FUNCTION_BLOCK PUBLIC EcMasterDeviceCount IMPLEMENTS IEcTask
VAR_INPUT
END_VAR
VAR_OUTPUT
END_VAR
VAR
	iState : INT;
	masterDeviceCount : Tc2_EtherCAT.FB_EcGetSlaveCount;
	_execute: BOOL;
	_done: BOOL;
	_busy: BOOL;
	_error: BOOL;
	_netId: AMSNETID;
END_VAR

CASE iState OF
	0:
		IF _execute THEN
			_done := FALSE;
			_busy := TRUE;
			_error := FALSE;
			masterDeviceCount.bExecute := TRUE;
			IF masterDeviceCount.bBusy THEN
				iState := 10;
				_execute := false;
			END_IF
		END_IF
	10:
		IF NOT masterDeviceCount.bBusy THEN
			IF NOT masterDeviceCount.bError THEN
				_done := TRUE;
			ELSE
				_error := TRUE;
			END_IF
			_busy := FALSE;
			masterDeviceCount.bExecute := FALSE;
			iState := 0;
		END_IF
END_CASE

masterDeviceCount(sNetId := Tc2_System.F_CreateAmsNetId(nIds := NetId));

{warning 'add method implementation '}
METHOD Abort : BOOL
masterDeviceCount.bExecute := FALSE;
_busy := FALSE;
_execute := FALSE;
Abort := TRUE;
iState := 0;
END_METHOD

{warning 'add property implementation'}
PROPERTY Busy : BOOL
GET
Busy := _busy;
END_GET
END_PROPERTY

{warning 'add property implementation'}
PROPERTY Done : BOOL
GET
Done := _done;
END_GET
END_PROPERTY

{warning 'add property implementation'}
PROPERTY Error : BOOL
GET
Error := _error;
END_GET
END_PROPERTY

METHOD Execute : BOOL
VAR_INPUT
END_VAR
IF NOT Busy THEN
	Execute := _execute := TRUE;
END_IF
END_METHOD

{warning 'add property implementation'}
PROPERTY NetID : amsnetid
GET
NetID := _netId;
END_GET
SET
_netId := NetID;
END_SET
END_PROPERTY

PROPERTY NumberDevices : uint
GET
NumberDevices := masterDeviceCount.nSlaves;
END_GET
END_PROPERTY

END_FUNCTION_BLOCK

(* stored: Version 1.1.0.1, ProductVersion 3.1.4024.11
   POU EcMasterDeviceCount: Id {fc00524b-5402-4693-86e9-fa947a8c9c97}, SpecialFunc None
   Method Abort: Id {3bae2c62-e9a5-46f5-ae36-84b500f63c8f}
   Property Busy: Id {65b26ac7-ba6c-4704-8ca8-eaff044310bf}
   Get Get: Id {a3bee638-4503-4be6-b6c3-fe7708296811}
   Property Done: Id {2c123594-83aa-4b23-821b-5ffde7c84b56}
   Get Get: Id {1f6b99bd-4106-4b36-8963-651a31143e8d}
   Property Error: Id {c2a38a2c-d091-482a-97fb-36810d338b20}
   Get Get: Id {1f539981-a3c3-4c3d-a4f1-1542bc59818d}
   Method Execute: Id {36d0869b-cbde-49a1-83fa-b9df4813c9b6}
   Property NetID: Id {14f9c1e4-a35b-43cc-84da-1c0e7fcdf0c9}
   Get Get: Id {925b4353-ca71-4dca-aa79-78985a9f6224}
   Set Set: Id {5dc8bdd8-1778-4212-bd96-63f763dc5f6f}
   Property NumberDevices: Id {0c16f1b3-a1d9-428e-8968-f6e24f86aafb}
   Get Get: Id {2e87b82c-875e-41f1-8552-6634c057e6cf} *)
